{attribute 'GeneratedUsingTerminal: EK1960-0000-0019'}
{attribute addProperty BoxType "EK1960-0000-0019"}
{attribute addProperty Id "FSoE_InputsFSoE_Inputs_9283FC6947FSoE_OutputsFSoE_Outputs_79E75DAB51"}
{attribute addProperty CRC "3197276151"}
{attribute addProperty Size "98"}
TYPE Module_1_FSoE_BE928FF7 :
STRUCT
	{attribute addProperty Name "FSoE_Inputs"}
	FSoE_Inputs  : FSoE_Inputs_9283FC69;
	{attribute addProperty Name "FSoE_Outputs"}
	FSoE_Outputs  : FSoE_Outputs_79E75DAB;
END_STRUCT
END_TYPE

(* stored: Version 1.2.0.0, ProductVersion 3.1.4024.9
   DUT Module_1_FSoE_BE928FF7: Id {0f9a5c7b-9ef7-44a9-8432-bd01efd0d858} *)
